TYPE T_Short_String : STRING(80); END_TYPE

(* stored: Version 1.1.0.1, ProductVersion 3.1.4024.4
   DUT T_Short_String: Id {26118e4f-060a-49c3-9e5e-6a6f465fb48a} *)
